{attribute 'call_after_init'}
FUNCTION_BLOCK FB_CarbideShutterEnable_Test EXTENDS FB_TestSuite
VAR_INPUT
END_VAR
VAR_OUTPUT
END_VAR
VAR
END_VAR

LocksWithHardwareFailure();
LocksWithLOCOLeak();
LocksWithLUTLeak();
EnablesWhenNoError();

METHOD EnablesWhenNoError
VAR
	stErrors : ST_ErrorStates;
	bResult : BOOL;
END_VAR
TEST('EnablesWhenNoErrors');

bResult := F_CarbideShutterEnable(stErrors := stErrors);

AssertTrue(bResult, 'Carbide Shutter did not enable');

TEST_FINISHED();
END_METHOD

METHOD LocksWithHardwareFailure
VAR
	stErrors : st_ErrorStates;
	bResult : BOOL;
END_VAR
TEST('LocksWithHardwareFailure');

stErrors.bHardwareFailure := TRUE;
bResult := F_CarbideShutterEnable(stErrors := stErrors);

AssertFalse(bResult, 'Carbide Shutter did not lock');

TEST_FINISHED();
END_METHOD

METHOD LocksWithLOCOLeak
VAR
	stErrors : st_ErrorStates;
	bResult : BOOL;
END_VAR
TEST('LocksWithLOCOLeak');

stErrors.bLeakOpcpaCarbideOn := TRUE;
bResult := F_CarbideShutterEnable(stErrors := stErrors);

AssertFalse(bResult, 'Carbide Shutter did not lock');

TEST_FINISHED();
END_METHOD

METHOD LocksWithLUTLeak
VAR
	stErrors : st_ErrorStates;
	bResult : BOOL;
END_VAR
TEST('LocksWithLUTLeak');

stErrors.bLeakUnderTable := TRUE;
bResult := F_CarbideShutterEnable(stErrors := stErrors);

AssertFalse(bResult, 'Carbide Shutter did not lock');

TEST_FINISHED();
END_METHOD

END_FUNCTION_BLOCK

(* stored: Version 1.1.0.1, ProductVersion 3.1.4022.17
   POU FB_CarbideShutterEnable_Test: Id {12de6daa-2e93-4cf6-a175-72c7908e4818}, SpecialFunc None
   Method EnablesWhenNoError: Id {d35f6819-3cc1-425c-b98c-a24d3a5c17ac}
   Method LocksWithHardwareFailure: Id {25e3c8ee-3140-46f3-988f-b8adec232a2e}
   Method LocksWithLOCOLeak: Id {3ffd3ee4-1739-44f7-84e6-c166e3dea094}
   Method LocksWithLUTLeak: Id {db1f4eaa-6df6-4aad-8499-aba8a84c8b8d} *)
